INTERFACE IPid

PROPERTY Out : LREAL
GET
END_GET
END_PROPERTY

END_INTERFACE

(* stored: Version 1.1.0.1, ProductVersion 3.1.4024.11
   Itf IPid: Id {8da9abfe-226e-4374-8b8c-042275335040}
   Property Out: Id {64068ae4-68b9-44bb-8ed8-fbb18b8f1488}
   Get Get: Id {9422e15c-8b73-4f5f-a681-6176ebc22db6} *)
